PROGRAM MAIN
VAR
	fbHigherLevel : HigherLevelFB;
	eException : E_Exception;
	stException : ST_Exception;
	
	bSystemException : BOOL;
	bLowPressureException : BOOL;
	bTestUnitWaitingForRelease : BOOL;
END_VAR

fbHigherLevel(eOrigin := eHIGHER_LEVEL);

IF fbHigherLevel.Receive(eWAIT_FOR_RELEASE_SIGNAL, eTEST_UNIT) 
THEN
	bTestUnitWaitingForRelease := TRUE;
END_IF

WHILE fbHigherLevel.ExceptionAvailable()
DO

	stException := fbHigherLevel.getException;
	
	CASE stException.eException OF
	
		eSYSTEM_EXCEPTION:
			//Stop machine operation for example
			bSystemException := TRUE;
			;
		eLOW_PRESSURE_EXCEPTION:
			bLowPressureException := TRUE;
			;
			
	END_CASE
	
END_WHILE

END_PROGRAM

(* stored: Version 1.1.0.1, ProductVersion 3.1.4024.0
   POU MAIN: Id {1169b5ad-787b-4637-95d4-2ca0401351eb}, SpecialFunc None *)
